{region '#Template'}
	{attribute 'Version' := '5.0.2.0'}
	{attribute 'Tags' := '"LCID": "1031", "Text": "Fassade, Sonnenschutz, Sturmschutz"'}
	{attribute 'Tags' := '"LCID": "1033", "Text": "Facade, Sunprotection, windprotection"'}
	{attribute 'Using' := '"Type": "Template", "URI": "ST_BA_SunBld"'}
	{attribute 'Using' := '"Type": "Template", "URI": "E_BA_SunBldPrio"'}
	{attribute 'Description' := '"LCID": "1031", "Text": "Sturmschutz"'}
	{attribute 'Description' := '"LCID": "1033", "Text": "Windprotection"'}
{endregion}
FUNCTION_BLOCK FB_BA_Facade_WindProtection EXTENDS FB_BA_View
VAR_INPUT
END_VAR
VAR_OUTPUT
	stSunbld					: ST_BA_SunBld;
	bWndPrtc					: BOOL;
	fWndSpdStormOn				: REAL;
	fWndSpdStormOff				: REAL;		
END_VAR
VAR_INPUT CONSTANT PERSISTENT	
	{attribute 'parameterUnit':= 'm/s'}
	aWndSpdLmtStormOn			: ARRAY[1..32] OF REAL;		// Storm-detection on-values for different directions
	{attribute 'parameterUnit':= 'm/s'}
	aWndSpdLmtStormOff			: ARRAY[1..32] OF REAL;		// Storm-detection off-values for different directions
END_VAR
VAR_INPUT CONSTANT
	DlyStrmOn					: FB_BA_AV_Op;		
	DlyStrmOff					: FB_BA_AV_Op;	
	WndPrtcState				: FB_BA_BV_Op;		
	SunBldWndPrtc				: FB_BA_SunBldWndPrtc;
END_VAR
VAR
	aStormDirection				: ARRAY[1..32] OF REAL :=	[0.0, 30.0, 60.0, 90.0, 120.0, 150.0, 180.0, 210.0, 240.0, 270.0, 300.0, 330.0, 360.0];
	StormOnInterpolation		: FB_BA_Chrct32;
	StormOffInterpolation		: FB_BA_Chrct32;
END_VAR

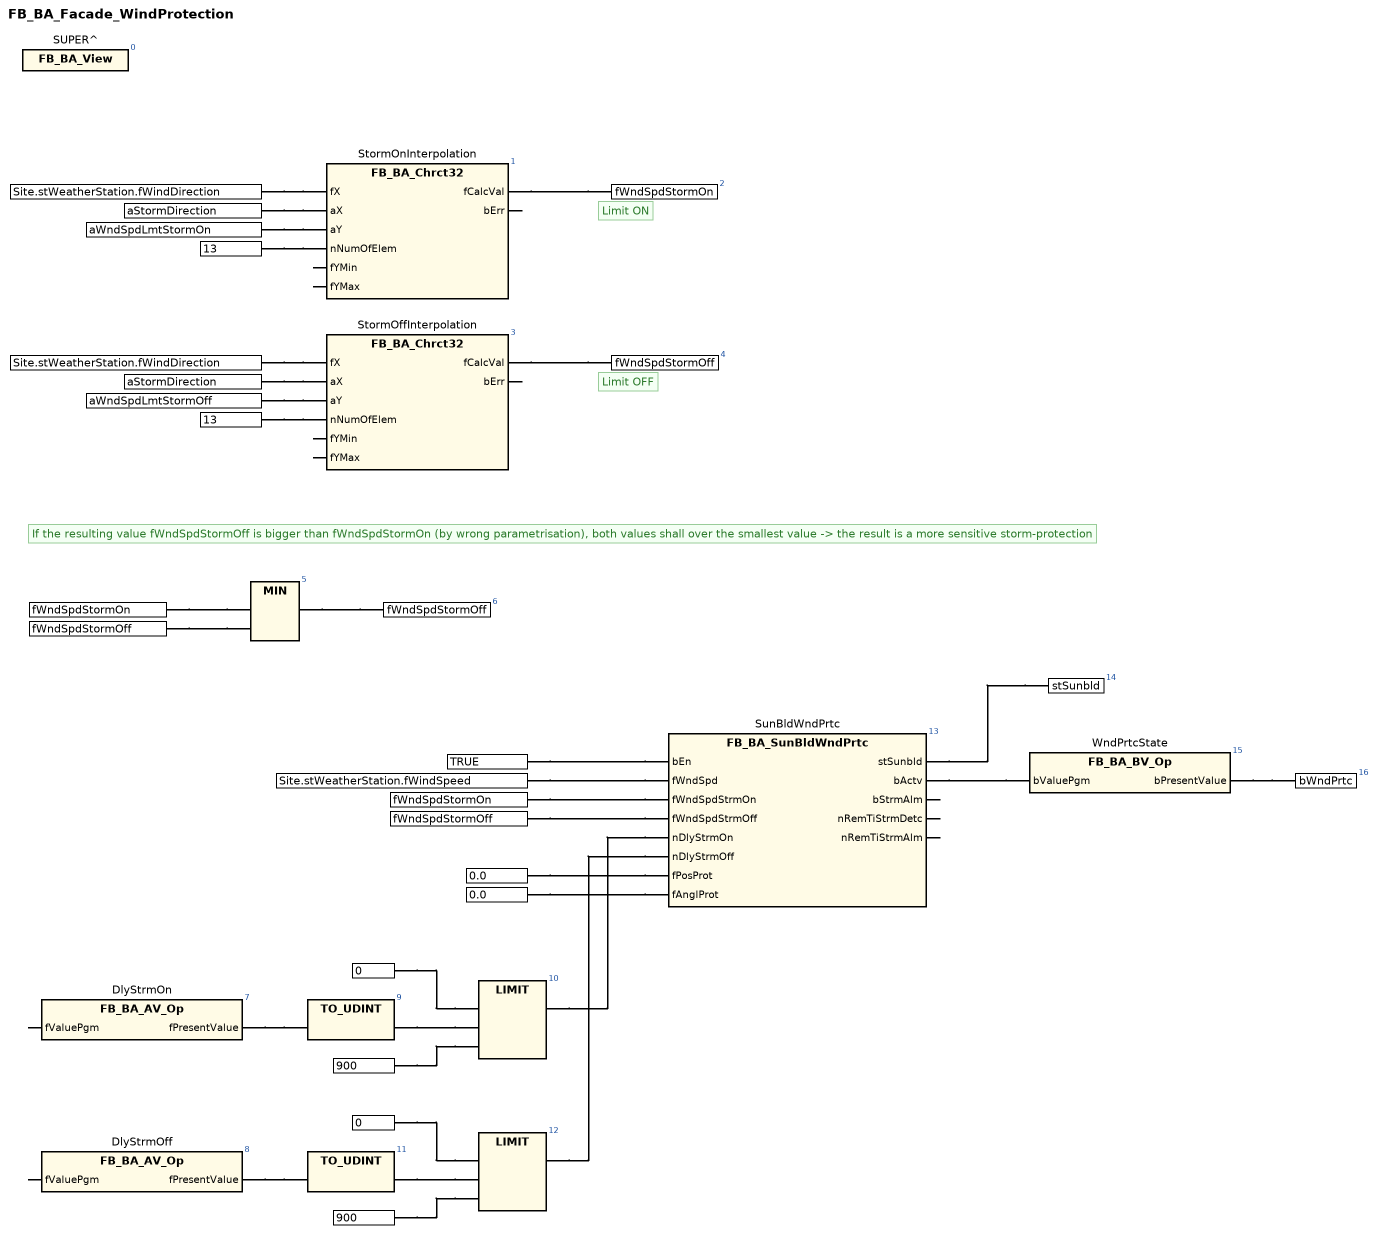
SUPER^(); // FB_BA_View
StormOnInterpolation(
    fX := Site.stWeatherStation.fWindDirection,
    aX := aStormDirection,
    aY := aWndSpdLmtStormOn,
    nNumOfElem := 13); // FB_BA_Chrct32
// Limit ON
fWndSpdStormOn := StormOnInterpolation.fCalcVal;
StormOffInterpolation(
    fX := Site.stWeatherStation.fWindDirection,
    aX := aStormDirection,
    aY := aWndSpdLmtStormOff,
    nNumOfElem := 13); // FB_BA_Chrct32
// Limit OFF
fWndSpdStormOff := StormOffInterpolation.fCalcVal;
// If the resulting value fWndSpdStormOff is bigger than fWndSpdStormOn (by wrong parametrisation), both values shall over the smallest value -> the result is a more sensitive storm-protection
fWndSpdStormOff := MIN(fWndSpdStormOn, fWndSpdStormOff);
DlyStrmOn(); // FB_BA_AV_Op
DlyStrmOff(); // FB_BA_AV_Op
SunBldWndPrtc(
    bEn := TRUE,
    fWndSpd := Site.stWeatherStation.fWindSpeed,
    fWndSpdStrmOn := fWndSpdStormOn,
    fWndSpdStrmOff := fWndSpdStormOff,
    nDlyStrmOn := LIMIT(0, TO_UDINT(DlyStrmOn.fPresentValue), 900),
    nDlyStrmOff := LIMIT(0, TO_UDINT(DlyStrmOff.fPresentValue), 900),
    fPosProt := 0.0,
    fAnglProt := 0.0); // FB_BA_SunBldWndPrtc
stSunbld := SunBldWndPrtc.stSunbld;
WndPrtcState(bValuePgm := SunBldWndPrtc.bActv); // FB_BA_BV_Op
bWndPrtc := WndPrtcState.bPresentValue;

METHOD FB_init : BOOL
VAR_INPUT
	bInitRetains : BOOL; // if TRUE; the retain variables are initialized (warm start / cold start)
	bInCopyCode : BOOL;  // if TRUE; the instance afterwards gets moved into the copy code (online change)
END_VAR
aWndSpdLmtStormOn[01]			:= 12;	// value [m/s] at 0 degree cardinal direction		// default value of 12 is in m/s and means "strong wind" - 6Bft
aWndSpdLmtStormOn[02]			:= 12;	// value [m/s] at 30 degree cardinal direction
aWndSpdLmtStormOn[03]			:= 12;	// value [m/s] at 60 degree cardinal direction
aWndSpdLmtStormOn[04]			:= 12;	// value [m/s] at 90 degree cardinal direction
aWndSpdLmtStormOn[05]			:= 12;	// value [m/s] at 120 degree cardinal direction
aWndSpdLmtStormOn[06]			:= 12;	// value [m/s] at 150 degree cardinal direction
aWndSpdLmtStormOn[07]			:= 12;	// value [m/s] at 180 degree cardinal direction
aWndSpdLmtStormOn[08]			:= 12;	// value [m/s] at 210 degree cardinal direction
aWndSpdLmtStormOn[09]			:= 12;	// value [m/s] at 240 degree cardinal direction
aWndSpdLmtStormOn[10]			:= 12;	// value [m/s] at 270 degree cardinal direction
aWndSpdLmtStormOn[11]			:= 12;	// value [m/s] at 300 degree cardinal direction
aWndSpdLmtStormOn[12]			:= 12;	// value [m/s] at 330 degree cardinal direction
aWndSpdLmtStormOn[13]			:= 12;	// value [m/s] at 360 degree cardinal direction

aWndSpdLmtStormOff[01]			:= 08;	// value [m/s] at 0 degree cardinal direction
aWndSpdLmtStormOff[02]			:= 08;	// value [m/s] at 30 degree cardinal direction
aWndSpdLmtStormOff[03]			:= 08;	// value [m/s] at 60 degree cardinal direction
aWndSpdLmtStormOff[04]			:= 08;	// value [m/s] at 90 degree cardinal direction
aWndSpdLmtStormOff[05]			:= 08;	// value [m/s] at 120 degree cardinal direction
aWndSpdLmtStormOff[06]			:= 08;	// value [m/s] at 150 degree cardinal direction
aWndSpdLmtStormOff[07]			:= 08;	// value [m/s] at 180 degree cardinal direction
aWndSpdLmtStormOff[08]			:= 08;	// value [m/s] at 210 degree cardinal direction
aWndSpdLmtStormOff[09]			:= 08;	// value [m/s] at 240 degree cardinal direction
aWndSpdLmtStormOff[10]			:= 08;	// value [m/s] at 270 degree cardinal direction
aWndSpdLmtStormOff[11]			:= 08;	// value [m/s] at 300 degree cardinal direction
aWndSpdLmtStormOff[12]			:= 08;	// value [m/s] at 330 degree cardinal direction
aWndSpdLmtStormOff[13]			:= 08;	// value [m/s] at 360 degree cardinal direction

DlyStrmOn.iParent				:= THIS^;
DlyStrmOn.iLabel				:= LblCtl_TimeDelayStormOn;
DlyStrmOn.sObjectName			:= '{Idx=01}';
DlyStrmOn.eUnit					:= E_BA_Unit.eTime_Seconds; 
DlyStrmOn.fValueRm				:= 10.0;
                       	
DlyStrmOff.iParent				:= THIS^;
DlyStrmOff.iLabel				:= LblCtl_TimeDelayStormOff;
DlyStrmOff.sObjectName			:= '{Idx=01}';
DlyStrmOff.eUnit				:= E_BA_Unit.eTime_Seconds; 
DlyStrmOff.fValueRm				:= 300.0;
                            	
WndPrtcState.iParent			:= THIS^;	
WndPrtcState.iLabel				:= LblCtl_WindProtectionState;
WndPrtcState.sObjectName		:= '{Idx=01}';
WndPrtcState.sInactiveText		:= txtEvent_Off;
WndPrtcState.sActiveText		:= txtEvent_On;
WndPrtcState.bValueRm			:= FALSE;								
WndPrtcState.eToggleMode 		:= E_BA_ToggleMode.eSwitch;
END_METHOD

END_FUNCTION_BLOCK

(* stored: Version 1.1.0.1, ProductVersion 3.1.4024.12
   POU FB_BA_Facade_WindProtection: Id {a11a43d6-605f-48b9-9db4-b002b2c6123c}, SpecialFunc None
   Method FB_init: Id {a8c6cf05-0b46-4fb9-bffa-cfc0d18b6443} *)
